(* IEC 61131-3 sources: AXOpen/src/components.ur.robotics/ctrl/src/AxoUrCb3 (part 2) *)

                    Outputs.MotorOn:=_blink.output;

                    IF Inputs.Inputs.Safety.FT_IsFault THEN
                        THIS.CallTimers(FALSE);
                        _power_progress := 310;
                    END_IF;

                    IF Inputs.Inputs.Robot.PW_IsPowerOn THEN
                         Outputs.MotorOn:=FALSE;
                         THIS.CallTimers(FALSE);
                         _power_progress := 321;
                    END_IF;
                END_IF;

                IF _power_progress = 321 THEN
                    TaskMessenger.ActivateOnCondition(ULINT#521, _infoTimer.output, eAxoMessageCategory#Warning);
                    IF _infoTimer.output THEN
                        RobotStatus.Error.Id := UINT#521;
                    END_IF;

                    Outputs.Start:=_blink.output;

                    IF Inputs.Inputs.Safety.FT_IsFault THEN
                        THIS.CallTimers(FALSE);
                        _power_progress := 310;
                    END_IF;

                    IF Inputs.Inputs.Robot.PR_IsProgramRunning AND NOT Inputs.Inputs.Safety.FT_IsFault THEN
                         Outputs.Start:=FALSE;
                         THIS.CallTimers(FALSE);
                         _power_progress := 322;
                    END_IF;
                END_IF;

                IF _power_progress = 322 THEN
                    StartMotorsAndProgramTask.DoneWhen(TRUE);
                    THIS.CallTimers(FALSE);
                    _power_progress := 0;
                END_IF;

                THIS.CallTimers(TRUE);
                StartMotorsAndProgramTask.ThrowWhen(_errorTimer.output);
                RobotStatus.Action.Id := TO_UINT(_power_progress);
            END_IF;
            IF StartMotorsAndProgramTask.DoneReached() THEN
                RobotStatus.Action.Id :=  UINT#111;
                RobotStatus.Error.Id :=  UINT#0;
            ELSIF StartMotorsAndProgramTask.ErrorOccured() THEN
                RobotStatus.Action.Id :=  UINT#810;
                RobotStatus.Error.Id  :=  UINT#810;
            ELSIF StartMotorsAndProgramTask.AbortTriggered() THEN
                RobotStatus.Action.Id :=  UINT#811;
                RobotStatus.Error.Id  :=  UINT#811;
            END_IF;
            Messenger.ActivateOnCondition(ULINT#810,StartMotorsAndProgramTask.HasError(), eAxoMessageCategory#Error);
            Messenger.ActivateOnCondition(ULINT#811,StartMotorsAndProgramTask.IsAborted(), eAxoMessageCategory#Error);
            Messenger.ActivateOnCondition(ULINT#112,StartMotorsAndProgramTask.RestoreTriggered() , eAxoMessageCategory#Error);
            IF StartMotorsAndProgramTask.RestoreTriggered() AND _power_progress >= 310 AND _power_progress <= 329  THEN
                RobotStatus.Action.Id :=  UINT#112;
                _power_progress := 0;
            END_IF;
            //*******************************************

            //***********StartMotorsProgramAndMovementsTask*******
            StartMotorsProgramAndMovementsTask.IsDisabled := _stopTasksAreActive OR StartProgramTask.IsBusy() OR StartMotorsTask.IsBusy() OR StartMovementsTask.IsBusy();
            IF StartMotorsProgramAndMovementsTask.StartTriggered() THEN
                RobotStatus.Action.Id :=  UINT#130;
            END_IF;
            Messenger.ActivateOnCondition(ULINT#130,StartMotorsProgramAndMovementsTask.IsBusy(), eAxoMessageCategory#Info);
            Messenger.ActivateOnCondition(ULINT#131,StartMotorsProgramAndMovementsTask.IsDone(), eAxoMessageCategory#Info);
            IF StartMotorsProgramAndMovementsTask.Execute() THEN
                _blink.Blink(Context := _context, inOnTime:=T#500MS,inOffTime:=T#500MS);

                IF _power_progress = 0 THEN
                    RobotStatus.Error.Id := UINT#0;
                    TaskMessenger.Restore();
                    THIS.CallTimers(FALSE);
                    _power_progress := 330;
                END_IF;

                IF _power_progress = 330 THEN
                    TaskMessenger.ActivateOnCondition(ULINT#530, _infoTimer.output AND NOT Inputs.Inputs.Safety.NO_IsNormalMode, eAxoMessageCategory#Warning);
                    TaskMessenger.ActivateOnCondition(ULINT#531, _infoTimer.output AND NOT Inputs.Inputs.Safety.RD_IsReducedMode, eAxoMessageCategory#Warning);
                    IF _infoTimer.output THEN
                        IF NOT Inputs.Inputs.Safety.NO_IsNormalMode THEN
                            RobotStatus.Error.Id := UINT#530;
                        END_IF;
                        IF NOT Inputs.Inputs.Safety.RD_IsReducedMode THEN
                            RobotStatus.Error.Id := UINT#531;
                        END_IF;
                    END_IF;

                    IF Inputs.Inputs.Safety.NO_IsNormalMode OR Inputs.Inputs.Safety.RD_IsReducedMode THEN
                        THIS.CallTimers(FALSE);
                        _power_progress:=332;
                    END_IF;
                END_IF;

                IF _power_progress = 332 THEN	//Reseting error
                    TaskMessenger.ActivateOnCondition(ULINT#632, _infoTimer.output, eAxoMessageCategory#Warning);
                    IF _infoTimer.output THEN
                        RobotStatus.Error.Id := UINT#632;
                    END_IF;

                    IF NOT Inputs.Inputs.Safety.FT_IsFault THEN
                        THIS.CallTimers(FALSE);
                        _power_progress := 333;
                    END_IF;
                END_IF;

                IF _power_progress = 333 THEN	//Reseting emergency stop error
                    TaskMessenger.ActivateOnCondition(ULINT#533, _infoTimer.output AND Inputs.Inputs.Safety.ES_IsEmergencyStopped , eAxoMessageCategory#Warning);
                    TaskMessenger.ActivateOnCondition(ULINT#534, _infoTimer.output AND Inputs.Inputs.Safety.PS_IsProtectiveStopped , eAxoMessageCategory#Warning);
                    TaskMessenger.ActivateOnCondition(ULINT#535, _infoTimer.output AND Inputs.Inputs.Safety.SS_IsSafeguardStopped , eAxoMessageCategory#Warning);
                    TaskMessenger.ActivateOnCondition(ULINT#536, _infoTimer.output AND Inputs.Inputs.Safety.RC_IsRecoveryMode , eAxoMessageCategory#Warning);
                    TaskMessenger.ActivateOnCondition(ULINT#537, _infoTimer.output AND Inputs.Inputs.Safety.ST_IsStoppedDueSafety , eAxoMessageCategory#Warning);
                    TaskMessenger.ActivateOnCondition(ULINT#538, _infoTimer.output AND Inputs.Inputs.Safety.VL_IsViolation , eAxoMessageCategory#Warning);
                    IF _infoTimer.output THEN
                        IF Inputs.Inputs.Safety.ES_IsEmergencyStopped  THEN
                            RobotStatus.Error.Id := UINT#533;
                        END_IF;
                        IF Inputs.Inputs.Safety.PS_IsProtectiveStopped  THEN
                            RobotStatus.Error.Id := UINT#534;
                        END_IF;
                        IF Inputs.Inputs.Safety.SS_IsSafeguardStopped  THEN
                            RobotStatus.Error.Id := UINT#535;
                        END_IF;
                        IF Inputs.Inputs.Safety.RC_IsRecoveryMode  THEN
                            RobotStatus.Error.Id := UINT#536;
                        END_IF;
                        IF Inputs.Inputs.Safety.ST_IsStoppedDueSafety  THEN
                            RobotStatus.Error.Id := UINT#537;
                        END_IF;
                        IF Inputs.Inputs.Safety.VL_IsViolation  THEN
                            RobotStatus.Error.Id := UINT#538;
                        END_IF;
                    END_IF;

                    IF NOT Inputs.Inputs.Safety.ES_IsEmergencyStopped
                        AND NOT Inputs.Inputs.Safety.PS_IsProtectiveStopped
                        AND NOT Inputs.Inputs.Safety.SS_IsSafeguardStopped
                        AND NOT Inputs.Inputs.Safety.RC_IsRecoveryMode
                        AND NOT Inputs.Inputs.Safety.ST_IsStoppedDueSafety
                        AND NOT Inputs.Inputs.Safety.VL_IsViolation THEN
                        THIS.CallTimers(FALSE);
                        _power_progress := 339;
                    END_IF;
                END_IF;

                IF _power_progress = 339 THEN	//Starting the motors
                    TaskMessenger.ActivateOnCondition(ULINT#539, _infoTimer.output, eAxoMessageCategory#Warning);
                    IF _infoTimer.output THEN
                        RobotStatus.Error.Id := UINT#539;
                    END_IF;

                    Outputs.MotorOn:=_blink.output;

                    IF Inputs.Inputs.Safety.FT_IsFault THEN
                        THIS.CallTimers(FALSE);
                        _power_progress := 330;
                    END_IF;

                    IF Inputs.Inputs.Robot.PW_IsPowerOn AND NOT Inputs.Inputs.Safety.FT_IsFault THEN
                         Outputs.MotorOn:=FALSE;
                         THIS.CallTimers(FALSE);
                         _power_progress := 340;
                    END_IF;
                END_IF;

                IF _power_progress = 340 THEN	// Starting the program
                    TaskMessenger.ActivateOnCondition(ULINT#540, _infoTimer.output, eAxoMessageCategory#Warning);
                    IF _infoTimer.output THEN
                        RobotStatus.Error.Id := UINT#540;
                    END_IF;

                    Outputs.Start:=_blink.output;

                    IF Inputs.Inputs.Safety.FT_IsFault THEN
                        THIS.CallTimers(FALSE);
                        _power_progress := 330;
                    END_IF;

                    IF Inputs.Inputs.Robot.PR_IsProgramRunning AND NOT Inputs.Inputs.Safety.FT_IsFault THEN
                         Outputs.Start:=FALSE;
                         THIS.CallTimers(FALSE);
                         _power_progress := 341;
                    END_IF;
                END_IF;

                IF _power_progress = 341 THEN // Setting the  movement parameters
                    TaskMessenger.ActivateOnCondition(ULINT#541, _infoTimer.output, eAxoMessageCategory#Warning);
                    IF _infoTimer.output THEN
                        RobotStatus.Error.Id := UINT#541;
                    END_IF;
                    Outputs.GlobalSpeed     := TO_DINT(RobotStatus.CurrentMovementParameters.GlobalSpeed);
                    Outputs.ToolNo          := TO_DINT(RobotStatus.CurrentMovementParameters.ToolNo);
                    Outputs.WorkobjectNo    := TO_DINT(RobotStatus.CurrentMovementParameters.WorkobjectNo);
                    Outputs.PointNo         := TO_DINT(RobotStatus.CurrentMovementParameters.PointNo);
                    Outputs.UserSpecSpeed1  := RobotStatus.CurrentMovementParameters.UserSpecSpeed1;
                    Outputs.UserSpecSpeed2  := RobotStatus.CurrentMovementParameters.UserSpecSpeed2;
                    Outputs.Coordinates     := RobotStatus.CurrentMovementParameters.Coordinates;

                    Outputs.ActionNo := DINT#254;

                    IF Outputs.ActionNo = Inputs.ActionNo THEN
                        THIS.CallTimers(FALSE);
                        _power_progress := 342;
                    END_IF;
                END_IF;

                IF _power_progress = 342 THEN //Comparing the movement parameters.
                    TaskMessenger.ActivateOnCondition(ULINT#542, _infoTimer.output AND Inputs.GlobalSpeed <> TO_DINT(RobotStatus.CurrentMovementParameters.GlobalSpeed), eAxoMessageCategory#Warning);
                    TaskMessenger.ActivateOnCondition(ULINT#543, _infoTimer.output AND Inputs.ToolNo <> TO_DINT(RobotStatus.CurrentMovementParameters.ToolNo), eAxoMessageCategory#Warning);
                    TaskMessenger.ActivateOnCondition(ULINT#544, _infoTimer.output AND Inputs.WorkobjectNo <> TO_DINT(RobotStatus.CurrentMovementParameters.WorkobjectNo), eAxoMessageCategory#Warning);
                    TaskMessenger.ActivateOnCondition(ULINT#545, _infoTimer.output AND Inputs.PointNo <> TO_DINT(RobotStatus.CurrentMovementParameters.PointNo), eAxoMessageCategory#Warning);
                    TaskMessenger.ActivateOnCondition(ULINT#546, _infoTimer.output AND Inputs.UserSpecSpeed1 <> RobotStatus.CurrentMovementParameters.UserSpecSpeed1, eAxoMessageCategory#Warning);
                    TaskMessenger.ActivateOnCondition(ULINT#547, _infoTimer.output AND Inputs.UserSpecSpeed2 <> RobotStatus.CurrentMovementParameters.UserSpecSpeed2, eAxoMessageCategory#Warning);
                    IF _infoTimer.output THEN
                        IF Inputs.GlobalSpeed <> TO_DINT(RobotStatus.CurrentMovementParameters.GlobalSpeed) THEN
                            RobotStatus.Error.Id := UINT#542;//<#Waiting for Inputs.GlobalSpeed to be equal to MovementParameters.GlobalSpeed!
                        END_IF;
                        IF Inputs.ToolNo <> TO_DINT(RobotStatus.CurrentMovementParameters.ToolNo) THEN
                            RobotStatus.Error.Id := UINT#543;//<#Waiting for Inputs.ToolNo to be equal to MovementParameters.ToolNo!
                        END_IF;
                        IF Inputs.WorkobjectNo <> TO_DINT(RobotStatus.CurrentMovementParameters.WorkobjectNo) THEN
                            RobotStatus.Error.Id := UINT#544;//<#Waiting for Inputs.WorkobjectNo to be equal to MovementParameters.WorkobjectNo!
                        END_IF;
                        IF Inputs.PointNo <> TO_DINT(RobotStatus.CurrentMovementParameters.PointNo) THEN
                            RobotStatus.Error.Id := UINT#545;//<#Waiting for Inputs.PointNo to be equal to MovementParameters.PointNo!
                        END_IF;
                        IF Inputs.UserSpecSpeed1 <> RobotStatus.CurrentMovementParameters.UserSpecSpeed1 THEN
                            RobotStatus.Error.Id := UINT#546;//<#Waiting for Inputs.UserSpecSpeed1 to be equal to MovementParameters.UserSpecSpeed1!
                        END_IF;
                        IF Inputs.UserSpecSpeed2 <> RobotStatus.CurrentMovementParameters.UserSpecSpeed2 THEN
                            RobotStatus.Error.Id := UINT#547;//<#Waiting for Inputs.UserSpecSpeed2 to be equal to MovementParameters.UserSpecSpeed2!
                        END_IF;
                    END_IF;

                    IF 	Inputs.GlobalSpeed      = TO_DINT(RobotStatus.CurrentMovementParameters.GlobalSpeed) AND
                        Inputs.ToolNo           = TO_DINT(RobotStatus.CurrentMovementParameters.ToolNo) AND
                        Inputs.WorkobjectNo     = TO_DINT(RobotStatus.CurrentMovementParameters.WorkobjectNo) AND
                        Inputs.PointNo          = TO_DINT(RobotStatus.CurrentMovementParameters.PointNo) AND
                        Inputs.UserSpecSpeed1   = RobotStatus.CurrentMovementParameters.UserSpecSpeed1 AND
                        Inputs.UserSpecSpeed2   = RobotStatus.CurrentMovementParameters.UserSpecSpeed2 AND
                        AXOpen.Components.Robotics.CoordinatesAreNearlyEqual(Inputs.Coordinates,RobotStatus.CurrentMovementParameters.Coordinates,REAL#0.01,REAL#0.01,REAL#0.01,REAL#0.01,REAL#0.01,REAL#0.01) THEN
                        THIS.CallTimers(FALSE);
                        _power_progress:=348;
                    END_IF;
                END_IF;

                IF _power_progress = 348 THEN //Acknowledging the movement parameters
                    TaskMessenger.ActivateOnCondition(ULINT#548, _infoTimer.output, eAxoMessageCategory#Warning);
                    IF _infoTimer.output THEN
                        RobotStatus.Error.Id := UINT#548;
                    END_IF;

                    Outputs.ActionNo := DINT#255;

                    IF Outputs.ActionNo = Inputs.ActionNo THEN
                        THIS.CallTimers(FALSE);
                        _power_progress:=349;
                    END_IF;
                END_IF;

                IF _power_progress = 349 THEN
                    TaskMessenger.ActivateOnCondition(ULINT#549, _infoTimer.output, eAxoMessageCategory#Warning);
                    IF _infoTimer.output THEN
                        RobotStatus.Error.Id := UINT#549;
                    END_IF;

                    Outputs.ActionNo := TO_DINT(RobotStatus.CurrentMovementParameters.ActionNo);

                    IF Outputs.ActionNo = Inputs.ActionNo THEN
                        THIS.CallTimers(FALSE);
                        _power_progress:=350;
                    END_IF;
                END_IF;

                IF _power_progress = 350 THEN
                    TaskMessenger.ActivateOnCondition(ULINT#550, _infoTimer.output, eAxoMessageCategory#Warning);
                    IF _infoTimer.output THEN
                        RobotStatus.Error.Id := UINT#550;
                    END_IF;

                    Outputs.ActionNo := DINT#255;

                    IF Outputs.ActionNo = Inputs.ActionNo THEN
                        _power_progress := 0;
                        StartMotorsProgramAndMovementsTask.DoneWhen(TRUE);
                    END_IF;
                END_IF;

	            THIS.CallTimers(TRUE);
                StartMotorsProgramAndMovementsTask.ThrowWhen(_errorTimer.output);
                RobotStatus.Action.Id := TO_UINT(_power_progress);
            END_IF;
            IF StartMotorsProgramAndMovementsTask.DoneReached() THEN
                RobotStatus.Action.Id :=  UINT#131;
                RobotStatus.Error.Id :=  UINT#0;
            ELSIF StartMotorsProgramAndMovementsTask.ErrorOccured() THEN
                RobotStatus.Action.Id :=  UINT#830;
                RobotStatus.Error.Id  :=  UINT#830;
            ELSIF StartMotorsProgramAndMovementsTask.AbortTriggered() THEN
                RobotStatus.Action.Id :=  UINT#831;
                RobotStatus.Error.Id  :=  UINT#831;
            END_IF;
            Messenger.ActivateOnCondition(ULINT#830,StartMotorsProgramAndMovementsTask.HasError(), eAxoMessageCategory#Error);
            Messenger.ActivateOnCondition(ULINT#831,StartMotorsProgramAndMovementsTask.IsAborted(), eAxoMessageCategory#Error);
            Messenger.ActivateOnCondition(ULINT#132,StartMotorsProgramAndMovementsTask.RestoreTriggered() , eAxoMessageCategory#Error);
            IF StartMotorsProgramAndMovementsTask.RestoreTriggered() AND _power_progress >= 330 AND _power_progress <= 359 THEN
                RobotStatus.Action.Id :=  UINT#132;
                _power_progress := 0;
            END_IF;
            //*******************************************

            //***********StartMotorsTask*****************
            StartMotorsTask.IsDisabled := _stopTasksAreActive OR StartMotorsProgramAndMovementsTask.IsBusy() OR StartMotorsAndProgramTask.IsBusy();
            IF StartMotorsTask.StartTriggered() THEN
                RobotStatus.Action.Id :=  UINT#160;
            END_IF;
            Messenger.ActivateOnCondition(ULINT#160,StartMotorsTask.IsBusy(), eAxoMessageCategory#Info);
            Messenger.ActivateOnCondition(ULINT#161,StartMotorsTask.IsDone(), eAxoMessageCategory#Info);
            IF StartMotorsTask.Execute() THEN
                _blink.Blink(Context := _context, inOnTime:=T#500MS,inOffTime:=T#500MS);

                IF _power_progress = 0 THEN
                    RobotStatus.Error.Id := UINT#0;
                    TaskMessenger.Restore();
                    THIS.CallTimers(FALSE);
                    _power_progress := 360;
                END_IF;

                IF _power_progress = 360 THEN
                    TaskMessenger.ActivateOnCondition(ULINT#560, _infoTimer.output AND NOT Inputs.Inputs.Safety.NO_IsNormalMode, eAxoMessageCategory#Warning);
                    TaskMessenger.ActivateOnCondition(ULINT#561, _infoTimer.output AND NOT Inputs.Inputs.Safety.RD_IsReducedMode, eAxoMessageCategory#Warning);
                    IF _infoTimer.output THEN
                        IF NOT Inputs.Inputs.Safety.NO_IsNormalMode THEN
                            RobotStatus.Error.Id := UINT#560;
                        END_IF;
                        IF NOT Inputs.Inputs.Safety.RD_IsReducedMode THEN
                            RobotStatus.Error.Id := UINT#561;
                        END_IF;
                    END_IF;

                    IF Inputs.Inputs.Safety.NO_IsNormalMode OR Inputs.Inputs.Safety.RD_IsReducedMode THEN
                        THIS.CallTimers(FALSE);
                        _power_progress:=362;
                    END_IF;

                END_IF;

                IF _power_progress = 362 THEN	//Reseting error
                    TaskMessenger.ActivateOnCondition(ULINT#562, _infoTimer.output, eAxoMessageCategory#Warning);

                    IF _infoTimer.output THEN
                        RobotStatus.Error.Id := UINT#562;
                    END_IF;

                    IF NOT Inputs.Inputs.Safety.FT_IsFault THEN
                        THIS.CallTimers(FALSE);
                        _power_progress := 363;
                    END_IF;
                END_IF;

                IF _power_progress = 363 THEN	//Reseting emergency stop error

                    TaskMessenger.ActivateOnCondition(ULINT#563, _infoTimer.output AND Inputs.Inputs.Safety.ES_IsEmergencyStopped , eAxoMessageCategory#Warning);
                    TaskMessenger.ActivateOnCondition(ULINT#564, _infoTimer.output AND Inputs.Inputs.Safety.PS_IsProtectiveStopped , eAxoMessageCategory#Warning);
                    TaskMessenger.ActivateOnCondition(ULINT#565, _infoTimer.output AND Inputs.Inputs.Safety.SS_IsSafeguardStopped , eAxoMessageCategory#Warning);
                    TaskMessenger.ActivateOnCondition(ULINT#566, _infoTimer.output AND Inputs.Inputs.Safety.RC_IsRecoveryMode , eAxoMessageCategory#Warning);
                    TaskMessenger.ActivateOnCondition(ULINT#567, _infoTimer.output AND Inputs.Inputs.Safety.ST_IsStoppedDueSafety , eAxoMessageCategory#Warning);
                    TaskMessenger.ActivateOnCondition(ULINT#568, _infoTimer.output AND Inputs.Inputs.Safety.VL_IsViolation , eAxoMessageCategory#Warning);
                    IF _infoTimer.output THEN
                        IF Inputs.Inputs.Safety.ES_IsEmergencyStopped  THEN
                            RobotStatus.Error.Id := UINT#563;
                        END_IF;
                        IF Inputs.Inputs.Safety.PS_IsProtectiveStopped  THEN
                            RobotStatus.Error.Id := UINT#564;
                        END_IF;
                        IF Inputs.Inputs.Safety.SS_IsSafeguardStopped  THEN
                            RobotStatus.Error.Id := UINT#565;
                        END_IF;
                        IF Inputs.Inputs.Safety.RC_IsRecoveryMode  THEN
                            RobotStatus.Error.Id := UINT#566;
                        END_IF;
                        IF Inputs.Inputs.Safety.ST_IsStoppedDueSafety  THEN
                            RobotStatus.Error.Id := UINT#567;
                        END_IF;
                        IF Inputs.Inputs.Safety.VL_IsViolation  THEN
                            RobotStatus.Error.Id := UINT#568;
                        END_IF;
                    END_IF;

                    IF NOT Inputs.Inputs.Safety.ES_IsEmergencyStopped
                        AND NOT Inputs.Inputs.Safety.PS_IsProtectiveStopped
                        AND NOT Inputs.Inputs.Safety.SS_IsSafeguardStopped
                        AND NOT Inputs.Inputs.Safety.RC_IsRecoveryMode
                        AND NOT Inputs.Inputs.Safety.ST_IsStoppedDueSafety
                        AND NOT Inputs.Inputs.Safety.VL_IsViolation THEN
                        THIS.CallTimers(FALSE);
                        _power_progress := 369;
                    END_IF;
                END_IF;

                IF _power_progress = 369 THEN
                    TaskMessenger.ActivateOnCondition(ULINT#569, _infoTimer.output AND NOT Inputs.Inputs.Robot.PW_IsPowerOn, eAxoMessageCategory#Warning);
                    TaskMessenger.ActivateOnCondition(ULINT#570, _infoTimer.output AND Inputs.Inputs.Safety.FT_IsFault, eAxoMessageCategory#Warning);
                    TaskMessenger.ActivateOnCondition(ULINT#571, _infoTimer.output AND Inputs.Inputs.Joints.JointMode_0 <> 253 , eAxoMessageCategory#Warning);
                    TaskMessenger.ActivateOnCondition(ULINT#572, _infoTimer.output AND Inputs.Inputs.Joints.JointMode_1 <> 253 , eAxoMessageCategory#Warning);
                    TaskMessenger.ActivateOnCondition(ULINT#573, _infoTimer.output AND Inputs.Inputs.Joints.JointMode_2 <> 253 , eAxoMessageCategory#Warning);
                    TaskMessenger.ActivateOnCondition(ULINT#574, _infoTimer.output AND Inputs.Inputs.Joints.JointMode_3 <> 253 , eAxoMessageCategory#Warning);
                    TaskMessenger.ActivateOnCondition(ULINT#575, _infoTimer.output AND Inputs.Inputs.Joints.JointMode_4 <> 253 , eAxoMessageCategory#Warning);
                    TaskMessenger.ActivateOnCondition(ULINT#576, _infoTimer.output AND Inputs.Inputs.Joints.JointMode_5 <> 253 , eAxoMessageCategory#Warning);

                    IF _infoTimer.output THEN
                        IF NOT Inputs.Inputs.Robot.PW_IsPowerOn THEN
                            RobotStatus.Error.Id := UINT#569;
                        END_IF;
                        IF Inputs.Inputs.Safety.FT_IsFault  THEN
                            RobotStatus.Error.Id := UINT#570;
                        END_IF;
                        IF Inputs.Inputs.Joints.JointMode_0 <> 253  THEN
                            RobotStatus.Error.Id := UINT#571;
                        END_IF;
                        IF Inputs.Inputs.Joints.JointMode_1 <> 253  THEN
                            RobotStatus.Error.Id := UINT#572;
                        END_IF;
                        IF Inputs.Inputs.Joints.JointMode_2 <> 253  THEN
                            RobotStatus.Error.Id := UINT#573;
                        END_IF;
                        IF Inputs.Inputs.Joints.JointMode_3 <> 253  THEN
                            RobotStatus.Error.Id := UINT#574;
                        END_IF;
                        IF Inputs.Inputs.Joints.JointMode_4 <> 253  THEN
                            RobotStatus.Error.Id := UINT#575;
                        END_IF;
                        IF Inputs.Inputs.Joints.JointMode_5 <> 253  THEN
                            RobotStatus.Error.Id := UINT#576;
                        END_IF;
                    END_IF;

                    Outputs.MotorOn:=_blink.output;

                    IF Inputs.Inputs.Safety.FT_IsFault THEN
                        THIS.CallTimers(FALSE);
                        _power_progress := 360;
                    END_IF;

                    IF Inputs.Inputs.Robot.PW_IsPowerOn AND NOT Inputs.Inputs.Safety.FT_IsFault  AND
                        Inputs.Inputs.Joints.JointMode_0 = 253 AND
                        Inputs.Inputs.Joints.JointMode_1 = 253 AND
                        Inputs.Inputs.Joints.JointMode_2 = 253 AND
                        Inputs.Inputs.Joints.JointMode_3 = 253 AND
                        Inputs.Inputs.Joints.JointMode_4 = 253 AND
                        Inputs.Inputs.Joints.JointMode_5 = 253 THEN
                         Outputs.MotorOn:=FALSE;
                         THIS.CallTimers(FALSE);
                         _power_progress := 377;
                    END_IF;
                END_IF;

                IF _power_progress = 377 THEN
                    StartMotorsTask.DoneWhen(TRUE);
                    THIS.CallTimers(FALSE);
                    _power_progress := 0;
                END_IF;

                THIS.CallTimers(TRUE);
                StartMotorsTask.ThrowWhen(_errorTimer.output);
                RobotStatus.Action.Id := TO_UINT(_power_progress);
            END_IF;
            IF StartMotorsTask.IsFirstExecutionCycle() THEN
                MovementParameters := RobotStatus.CurrentMovementParameters;
            END_IF;
            IF StartMotorsTask.DoneReached() THEN
                RobotStatus.Action.Id :=  UINT#161;
                RobotStatus.Error.Id :=  UINT#0;
            ELSIF StartMotorsTask.ErrorOccured() THEN
                RobotStatus.Action.Id :=  UINT#860;
                RobotStatus.Error.Id  :=  UINT#860;
            ELSIF StartMotorsTask.AbortTriggered() THEN
                RobotStatus.Action.Id :=  UINT#861;
                RobotStatus.Error.Id  :=  UINT#861;
            END_IF;
            Messenger.ActivateOnCondition(ULINT#860,StartMotorsTask.HasError(), eAxoMessageCategory#Error);
            Messenger.ActivateOnCondition(ULINT#861,StartMotorsTask.IsAborted(), eAxoMessageCategory#Error);
            Messenger.ActivateOnCondition(ULINT#162,StartMotorsTask.RestoreTriggered() , eAxoMessageCategory#Error);
            IF StartMotorsTask.RestoreTriggered() AND _power_progress >= 360 AND _power_progress <= 379 THEN
                RobotStatus.Action.Id :=  UINT#162;
                _power_progress := 0;
            END_IF;

            //*******************************************

            //***********StartMovementsTask**************
            StartMovementsTask.IsDisabled := _stopTasksAreActive OR StartMotorsProgramAndMovementsTask.IsBusy();
            IF StartMovementsTask.StartTriggered() THEN
                RobotStatus.Action.Id :=  UINT#180;
            END_IF;
            Messenger.ActivateOnCondition(ULINT#180,StartMovementsTask.IsBusy(), eAxoMessageCategory#Info);
            Messenger.ActivateOnCondition(ULINT#181,StartMovementsTask.IsDone(), eAxoMessageCategory#Info);
            IF StartMovementsTask.Execute() THEN
                IF _movement_progress = 0 THEN
                    RobotStatus.Error.Id :=  UINT#0;
                    TaskMessenger.Restore();
                    THIS.CallTimers(FALSE);
                    _movement_progress := 380;
                END_IF;

                IF _movement_progress = 380 THEN
                    TaskMessenger.ActivateOnCondition(ULINT#580, _infoTimer.output, eAxoMessageCategory#Warning);
                    IF _infoTimer.output THEN
                        RobotStatus.Error.Id := UINT#580;
                    END_IF;

                    IF Inputs.Inputs.Robot.PR_IsProgramRunning THEN
                        THIS.CallTimers(FALSE);
                        _movement_progress := 381;
                    END_IF;
                END_IF;

                IF _movement_progress = 381 THEN
                    TaskMessenger.ActivateOnCondition(ULINT#581, _infoTimer.output, eAxoMessageCategory#Warning);
                    IF _infoTimer.output THEN
                        RobotStatus.Error.Id := UINT#581;
                    END_IF;

                    IF Inputs.Inputs.Robot.PW_IsPowerOn THEN
                        THIS.CallTimers(FALSE);
                        _movement_progress := 382;
                    END_IF;
                END_IF;

                IF _movement_progress = 382 THEN
                    TaskMessenger.ActivateOnCondition(ULINT#582, _infoTimer.output, eAxoMessageCategory#Warning);
                    IF _infoTimer.output THEN
                        RobotStatus.Error.Id := UINT#582;
                    END_IF;

                    IF NOT Inputs.Inputs.Safety.FT_IsFault THEN
                        THIS.CallTimers(FALSE);
                        _movement_progress := 383;
                    END_IF;
                END_IF;

                IF _movement_progress = 383 THEN
                    TaskMessenger.ActivateOnCondition(ULINT#583, _infoTimer.output, eAxoMessageCategory#Warning);
                    IF _infoTimer.output THEN
                        RobotStatus.Error.Id := UINT#583;
                    END_IF;

                    Outputs.GlobalSpeed     := TO_DINT(RobotStatus.CurrentMovementParameters.GlobalSpeed);
                    Outputs.ToolNo          := TO_DINT(RobotStatus.CurrentMovementParameters.ToolNo);
                    Outputs.WorkobjectNo    := TO_DINT(RobotStatus.CurrentMovementParameters.WorkobjectNo);
                    Outputs.PointNo         := TO_DINT(RobotStatus.CurrentMovementParameters.PointNo);
                    Outputs.UserSpecSpeed1  := RobotStatus.CurrentMovementParameters.UserSpecSpeed1;
                    Outputs.UserSpecSpeed2  := RobotStatus.CurrentMovementParameters.UserSpecSpeed2;
                    Outputs.Coordinates     := RobotStatus.CurrentMovementParameters.Coordinates;

                    Outputs.ActionNo := DINT#254;

                    IF Outputs.ActionNo = Inputs.ActionNo THEN
                        THIS.CallTimers(FALSE);
                        _power_progress := 384;
                    END_IF;
                END_IF;

                IF _power_progress = 384 THEN
                    TaskMessenger.ActivateOnCondition(ULINT#584, _infoTimer.output AND Inputs.GlobalSpeed <> TO_DINT(RobotStatus.CurrentMovementParameters.GlobalSpeed), eAxoMessageCategory#Warning);
                    TaskMessenger.ActivateOnCondition(ULINT#585, _infoTimer.output AND Inputs.ToolNo <> TO_DINT(RobotStatus.CurrentMovementParameters.ToolNo), eAxoMessageCategory#Warning);
                    TaskMessenger.ActivateOnCondition(ULINT#586, _infoTimer.output AND Inputs.WorkobjectNo <> TO_DINT(RobotStatus.CurrentMovementParameters.WorkobjectNo) , eAxoMessageCategory#Warning);
                    TaskMessenger.ActivateOnCondition(ULINT#587, _infoTimer.output AND Inputs.PointNo <> TO_DINT(RobotStatus.CurrentMovementParameters.PointNo) , eAxoMessageCategory#Warning);
                    TaskMessenger.ActivateOnCondition(ULINT#588, _infoTimer.output AND Inputs.UserSpecSpeed1 <> RobotStatus.CurrentMovementParameters.UserSpecSpeed1 , eAxoMessageCategory#Warning);
                    TaskMessenger.ActivateOnCondition(ULINT#589, _infoTimer.output AND Inputs.UserSpecSpeed2 <> RobotStatus.CurrentMovementParameters.UserSpecSpeed2, eAxoMessageCategory#Warning);

                    IF _infoTimer.output THEN
                        IF Inputs.GlobalSpeed <> TO_DINT(RobotStatus.CurrentMovementParameters.GlobalSpeed) THEN
                            RobotStatus.Error.Id := UINT#584;//<#Waiting for Inputs.GlobalSpeed to be equal to MovementParameters.GlobalSpeed!
                        END_IF;
                        IF Inputs.ToolNo <> TO_DINT(RobotStatus.CurrentMovementParameters.ToolNo) THEN
                            RobotStatus.Error.Id := UINT#585;//<#Waiting for Inputs.ToolNo to be equal to MovementParameters.ToolNo!
                        END_IF;
                        IF Inputs.WorkobjectNo <> TO_DINT(RobotStatus.CurrentMovementParameters.WorkobjectNo) THEN
                            RobotStatus.Error.Id := UINT#586;//<#Waiting for Inputs.WorkobjectNo to be equal to MovementParameters.WorkobjectNo!
                        END_IF;
                        IF Inputs.PointNo <> TO_DINT(RobotStatus.CurrentMovementParameters.PointNo) THEN
                            RobotStatus.Error.Id := UINT#587;//<#Waiting for Inputs.PointNo to be equal to MovementParameters.PointNo!
                        END_IF;
                        IF Inputs.UserSpecSpeed1 <> RobotStatus.CurrentMovementParameters.UserSpecSpeed1 THEN
                            RobotStatus.Error.Id := UINT#588;//<#Waiting for Inputs.UserSpecSpeed1 to be equal to MovementParameters.UserSpecSpeed1!
                        END_IF;
                        IF Inputs.UserSpecSpeed2 <> RobotStatus.CurrentMovementParameters.UserSpecSpeed2 THEN
                            RobotStatus.Error.Id := UINT#589;//<#Waiting for Inputs.UserSpecSpeed2 to be equal to MovementParameters.UserSpecSpeed2!
                        END_IF;
                    END_IF;

                    IF 	Inputs.GlobalSpeed      = TO_DINT(RobotStatus.CurrentMovementParameters.GlobalSpeed) AND
                        Inputs.ToolNo           = TO_DINT(RobotStatus.CurrentMovementParameters.ToolNo) AND
                        Inputs.WorkobjectNo     = TO_DINT(RobotStatus.CurrentMovementParameters.WorkobjectNo) AND
                        Inputs.PointNo          = TO_DINT(RobotStatus.CurrentMovementParameters.PointNo) AND
                        Inputs.UserSpecSpeed1   = RobotStatus.CurrentMovementParameters.UserSpecSpeed1 AND
                        Inputs.UserSpecSpeed2   = RobotStatus.CurrentMovementParameters.UserSpecSpeed2 AND
                        AXOpen.Components.Robotics.CoordinatesAreNearlyEqual(Inputs.Coordinates,RobotStatus.CurrentMovementParameters.Coordinates,REAL#0.01,REAL#0.01,REAL#0.01,REAL#0.01,REAL#0.01,REAL#0.01) THEN
                        THIS.CallTimers(FALSE);
                        _movement_progress:=390;
                    END_IF;
                END_IF;

                IF _movement_progress = 390 THEN
                    TaskMessenger.ActivateOnCondition(ULINT#590, _infoTimer.output, eAxoMessageCategory#Warning);
                    IF _infoTimer.output THEN
                        RobotStatus.Error.Id := UINT#590;
                    END_IF;

                    Outputs.ActionNo := DINT#255;

                    IF Outputs.ActionNo = Inputs.ActionNo THEN
                        THIS.CallTimers(FALSE);
                        _movement_progress:=391;
                    END_IF;
                END_IF;

                IF _movement_progress = 391 THEN
                    TaskMessenger.ActivateOnCondition(ULINT#591, _infoTimer.output, eAxoMessageCategory#Warning);
                    IF _infoTimer.output THEN
                        RobotStatus.Error.Id := UINT#591;
                    END_IF;

                    Outputs.ActionNo := TO_DINT(RobotStatus.CurrentMovementParameters.ActionNo);

                    IF Outputs.ActionNo = Inputs.ActionNo THEN
                        THIS.CallTimers(FALSE);
                        _movement_progress:=392;
                    END_IF;
                END_IF;

                IF _movement_progress = 392 THEN
                    TaskMessenger.ActivateOnCondition(ULINT#692, _infoTimer.output, eAxoMessageCategory#Warning);
                    IF _infoTimer.output THEN
                        RobotStatus.Error.Id := UINT#692;
                    END_IF;

                    Outputs.ActionNo := DINT#255;

                    IF Outputs.ActionNo = Inputs.ActionNo THEN
                        _movement_progress := 0;
                        StartMovementsTask.DoneWhen(TRUE);
                    END_IF;
                END_IF;

	            THIS.CallTimers(TRUE);

                StartMovementsTask.ThrowWhen(_errorTimer.output);

                RobotStatus.Action.Id := TO_UINT(_movement_progress);
            END_IF;
            IF StartMovementsTask.DoneReached() THEN
                RobotStatus.Action.Id :=  UINT#181;
                RobotStatus.Error.Id :=  UINT#0;
            ELSIF StartMovementsTask.ErrorOccured() THEN
                RobotStatus.Action.Id :=  UINT#880;
                RobotStatus.Error.Id  :=  UINT#880;
            ELSIF StartMovementsTask.AbortTriggered()THEN
                RobotStatus.Action.Id :=  UINT#881;
                RobotStatus.Error.Id  :=  UINT#881;
            END_IF;
            Messenger.ActivateOnCondition(ULINT#880,StartMovementsTask.HasError(), eAxoMessageCategory#Error);
            Messenger.ActivateOnCondition(ULINT#881,StartMovementsTask.IsAborted(), eAxoMessageCategory#Error);
            Messenger.ActivateOnCondition(ULINT#182,StartMovementsTask.RestoreTriggered() , eAxoMessageCategory#Error);
            IF StartMovementsTask.RestoreTriggered() AND _movement_progress >= 380 AND _movement_progress <= 399  THEN
                RobotStatus.Action.Id :=  UINT#182;
                _movement_progress := 0;
            END_IF;

            //*******************************************

            //***********StartProgramTask*******
            StartProgramTask.IsDisabled := _stopTasksAreActive;
            IF StartProgramTask.StartTriggered() THEN
                RobotStatus.Action.Id :=  UINT#200;
            END_IF;
            Messenger.ActivateOnCondition(ULINT#200,StartProgramTask.IsBusy(), eAxoMessageCategory#Info);
            Messenger.ActivateOnCondition(ULINT#201,StartProgramTask.IsDone(), eAxoMessageCategory#Info);
             IF StartProgramTask.Execute() THEN
                _blink.Blink(Context := _context, inOnTime:=T#500MS,inOffTime:=T#500MS);

                IF _power_progress = 0 THEN
                    RobotStatus.Error.Id :=  UINT#0;
                    TaskMessenger.Restore();
                    THIS.CallTimers(FALSE);
                    _power_progress := 400;
                END_IF;

                IF _power_progress = 400 THEN
                    TaskMessenger.ActivateOnCondition(ULINT#600, _infoTimer.output AND NOT Inputs.Inputs.Safety.NO_IsNormalMode, eAxoMessageCategory#Warning);
                    TaskMessenger.ActivateOnCondition(ULINT#601, _infoTimer.output AND NOT Inputs.Inputs.Safety.RD_IsReducedMode, eAxoMessageCategory#Warning);
                    IF _infoTimer.output THEN
                        IF NOT Inputs.Inputs.Safety.NO_IsNormalMode THEN
                            RobotStatus.Error.Id := UINT#600;
                        END_IF;
                        IF NOT Inputs.Inputs.Safety.RD_IsReducedMode THEN
                            RobotStatus.Error.Id := UINT#601;
                        END_IF;
                    END_IF;

                    IF Inputs.Inputs.Safety.NO_IsNormalMode OR Inputs.Inputs.Safety.RD_IsReducedMode THEN
                        THIS.CallTimers(FALSE);
                        _power_progress:=402;
                    END_IF;
                END_IF;

                IF _power_progress = 402 THEN
                    TaskMessenger.ActivateOnCondition(ULINT#602, _infoTimer.output, eAxoMessageCategory#Warning);
                    IF _infoTimer.output THEN
                        RobotStatus.Error.Id := UINT#602;
                    END_IF;

                    Outputs.Start:=_blink.output;

                    IF Inputs.Inputs.Robot.PR_IsProgramRunning THEN
                         Outputs.Start:=FALSE;
                         THIS.CallTimers(FALSE);
                         _power_progress := 403;
                    END_IF;
                END_IF;

                IF _power_progress = 403 THEN
                    StartProgramTask.DoneWhen(TRUE);
                    THIS.CallTimers(FALSE);
                    _power_progress := 0;
                END_IF;

                THIS.CallTimers(TRUE);
                StartProgramTask.ThrowWhen(_errorTimer.output);
                RobotStatus.Action.Id := TO_UINT(_power_progress);
            END_IF;
            IF StartProgramTask.DoneReached() THEN
                RobotStatus.Action.Id :=  UINT#201;
                RobotStatus.Error.Id :=  UINT#0;
            ELSIF StartProgramTask.ErrorOccured() THEN
                RobotStatus.Action.Id :=  UINT#900;
                RobotStatus.Error.Id  :=  UINT#900;
            ELSIF StartProgramTask.AbortTriggered()THEN
                RobotStatus.Action.Id :=  UINT#901;
                RobotStatus.Error.Id  :=  UINT#901;
            END_IF;
            Messenger.ActivateOnCondition(ULINT#900,StartProgramTask.HasError(), eAxoMessageCategory#Error);
            Messenger.ActivateOnCondition(ULINT#901,StartProgramTask.IsAborted(), eAxoMessageCategory#Error);
            Messenger.ActivateOnCondition(ULINT#202,StartProgramTask.RestoreTriggered() , eAxoMessageCategory#Error);
            IF StartProgramTask.RestoreTriggered() AND _power_progress >= 400 AND _power_progress <= 409  THEN
                RobotStatus.Action.Id :=  UINT#202;
                _power_progress := 0;
            END_IF;
            //*******************************************

            //***********StopMovementsAndProgramTask*****
            StopMovementsAndProgramTask.IsDisabled := FALSE;
            IF StopMovementsAndProgramTask.StartTriggered() THEN
                RobotStatus.Action.Id :=  UINT#210;
            END_IF;
            Messenger.ActivateOnCondition(ULINT#210,StopMovementsAndProgramTask.IsBusy(), eAxoMessageCategory#Info);
            Messenger.ActivateOnCondition(ULINT#211,StopMovementsAndProgramTask.IsDone(), eAxoMessageCategory#Info);
            IF StopMovementsAndProgramTask.Execute() THEN
                IF _power_progress = 0 THEN
                    RobotStatus.Error.Id :=  UINT#0;
                    TaskMessenger.Restore();
                    THIS.CallTimers(FALSE);
                    _power_progress := 410;
                END_IF;

                IF _power_progress = 410 THEN
                    TaskMessenger.ActivateOnCondition(ULINT#610, _infoTimer.output AND NOT Inputs.Inputs.Safety.NO_IsNormalMode, eAxoMessageCategory#Warning);
                    TaskMessenger.ActivateOnCondition(ULINT#611, _infoTimer.output AND NOT Inputs.Inputs.Safety.RD_IsReducedMode, eAxoMessageCategory#Warning);
                    IF _infoTimer.output THEN
                        IF NOT Inputs.Inputs.Safety.NO_IsNormalMode THEN
                            RobotStatus.Error.Id := UINT#610;
                        END_IF;
                        IF NOT Inputs.Inputs.Safety.RD_IsReducedMode THEN
                            RobotStatus.Error.Id := UINT#611;
                        END_IF;
                    END_IF;

                    IF Inputs.Inputs.Safety.NO_IsNormalMode OR Inputs.Inputs.Safety.RD_IsReducedMode THEN
                        THIS.CallTimers(FALSE);
                        _power_progress:=412;
                    END_IF;
                END_IF;

                IF _power_progress = 412 THEN
                    TaskMessenger.ActivateOnCondition(ULINT#612, _infoTimer.output, eAxoMessageCategory#Warning);
                    IF _infoTimer.output THEN
                        RobotStatus.Error.Id := UINT#612;
                    END_IF;

                    Outputs.Stop := TRUE;

                    IF NOT Inputs.Inputs.Robot.PR_IsProgramRunning THEN
                        Outputs.Stop := FALSE ;
                        THIS.CallTimers(FALSE);
                        _power_progress:=413;
                    END_IF;
                END_IF;

                IF _power_progress = 413 THEN
                    Outputs.Pause := FALSE ;
                    StopMovementsAndProgramTask.DoneWhen(TRUE);
                    _power_progress := 0;
                END_IF;

                THIS.CallTimers(TRUE);

                StopMovementsAndProgramTask.ThrowWhen(_errorTimer.output);

                RobotStatus.Action.Id := TO_UINT(_power_progress);
            END_IF;
            IF StopMovementsAndProgramTask.DoneReached() THEN
                RobotStatus.Action.Id :=  UINT#211;
                RobotStatus.Error.Id :=  UINT#0;
            ELSIF StopMovementsAndProgramTask.ErrorOccured() THEN
                RobotStatus.Action.Id :=  UINT#910;
                RobotStatus.Error.Id  :=  UINT#910;
            ELSIF StopMovementsAndProgramTask.AbortTriggered()THEN
                RobotStatus.Action.Id :=  UINT#911;
                RobotStatus.Error.Id  :=  UINT#911;
            END_IF;
            Messenger.ActivateOnCondition(ULINT#910,StopMovementsAndProgramTask.HasError(), eAxoMessageCategory#Error);
            Messenger.ActivateOnCondition(ULINT#911,StopMovementsAndProgramTask.IsAborted(), eAxoMessageCategory#Error);
            Messenger.ActivateOnCondition(ULINT#212,StopMovementsAndProgramTask.RestoreTriggered() , eAxoMessageCategory#Error);
            IF StopMovementsAndProgramTask.RestoreTriggered() AND _power_progress >= 410 AND _power_progress <= 419  THEN
                RobotStatus.Action.Id :=  UINT#212;
                _power_progress := 0;
            END_IF;
            //*******************************************

            //***********StopMovementsTask***************
            StopMovementsTask.IsDisabled := FALSE;
            IF StopMovementsAndProgramTask.StartTriggered() THEN
                RobotStatus.Action.Id :=  UINT#220;
            END_IF;
            Messenger.ActivateOnCondition(ULINT#220,StopMovementsAndProgramTask.IsBusy(), eAxoMessageCategory#Info);
            Messenger.ActivateOnCondition(ULINT#221,StopMovementsAndProgramTask.IsDone(), eAxoMessageCategory#Info);
            IF StopMovementsTask.Execute() THEN
                IF _power_progress = 0 THEN
                    RobotStatus.Error.Id :=  UINT#0;
                    TaskMessenger.Restore();
                    THIS.CallTimers(FALSE);
                    _power_progress := 420;
                END_IF;

                IF _power_progress = 420 THEN
                    TaskMessenger.ActivateOnCondition(ULINT#620, _infoTimer.output AND NOT Inputs.Inputs.Safety.NO_IsNormalMode, eAxoMessageCategory#Warning);
                    TaskMessenger.ActivateOnCondition(ULINT#621, _infoTimer.output AND NOT Inputs.Inputs.Safety.RD_IsReducedMode, eAxoMessageCategory#Warning);
                    IF _infoTimer.output THEN
                        IF NOT Inputs.Inputs.Safety.NO_IsNormalMode THEN
                            RobotStatus.Error.Id := UINT#620;
                        END_IF;
                        IF NOT Inputs.Inputs.Safety.RD_IsReducedMode THEN
                            RobotStatus.Error.Id := UINT#621;
                        END_IF;
                    END_IF;

                    IF Inputs.Inputs.Safety.NO_IsNormalMode OR Inputs.Inputs.Safety.RD_IsReducedMode THEN
                        THIS.CallTimers(FALSE);
                        _power_progress:=422;
                    END_IF;
                END_IF;
                IF _power_progress = 422 THEN
                    TaskMessenger.ActivateOnCondition(ULINT#622, _infoTimer.output, eAxoMessageCategory#Warning);
                    IF _infoTimer.output THEN
                        RobotStatus.Error.Id := UINT#622;
                    END_IF;

                    Outputs.Pause := TRUE;

                    IF NOT Inputs.Inputs.Robot.PR_IsProgramRunning THEN
                        Outputs.Pause := FALSE ;
                        THIS.CallTimers(FALSE);
                        _power_progress:=423;
                    END_IF;
                END_IF;

                IF _power_progress = 423 THEN
                    Outputs.Pause := FALSE ;
                    StopMovementsTask.DoneWhen(TRUE);
                    _power_progress := 0;
                END_IF;
                THIS.CallTimers(TRUE);

                StopMovementsTask.ThrowWhen(_errorTimer.output);

                RobotStatus.Action.Id := TO_UINT(_power_progress);
            END_IF;
            IF StopMovementsTask.DoneReached() THEN
                RobotStatus.Action.Id :=  UINT#221;
                RobotStatus.Error.Id :=  UINT#0;
            ELSIF StopMovementsTask.ErrorOccured() THEN
                RobotStatus.Action.Id :=  UINT#920;
                RobotStatus.Error.Id  :=  UINT#920;
            ELSIF StopMovementsTask.AbortTriggered()THEN
                RobotStatus.Action.Id :=  UINT#921;
                RobotStatus.Error.Id  :=  UINT#921;
            END_IF;
            Messenger.ActivateOnCondition(ULINT#920,StopMovementsTask.HasError(), eAxoMessageCategory#Error);
            Messenger.ActivateOnCondition(ULINT#921,StopMovementsTask.IsAborted(), eAxoMessageCategory#Error);
            Messenger.ActivateOnCondition(ULINT#222,StopMovementsTask.RestoreTriggered() , eAxoMessageCategory#Error);
            IF StopMovementsTask.RestoreTriggered() AND _power_progress >= 420 AND _power_progress <= 429  THEN
                RobotStatus.Action.Id :=  UINT#222;
                _power_progress := 0;
            END_IF;
            //*******************************************

            //***********StopProgramTask*****************
            StopProgramTask.IsDisabled := FALSE;
            IF StopProgramTask.StartTriggered() THEN
                RobotStatus.Action.Id :=  UINT#230;
            END_IF;
            Messenger.ActivateOnCondition(ULINT#230,StopProgramTask.IsBusy(), eAxoMessageCategory#Info);
            Messenger.ActivateOnCondition(ULINT#231,StopProgramTask.IsDone(), eAxoMessageCategory#Info);
            IF StopProgramTask.Execute() THEN
                IF _power_progress = 0 THEN
                    RobotStatus.Error.Id :=  UINT#0;
                    TaskMessenger.Restore();
                    THIS.CallTimers(FALSE);
                    _power_progress := 430;
                END_IF;

                IF _power_progress = 430 THEN
                    TaskMessenger.ActivateOnCondition(ULINT#630, _infoTimer.output AND NOT Inputs.Inputs.Safety.NO_IsNormalMode, eAxoMessageCategory#Warning);
                    TaskMessenger.ActivateOnCondition(ULINT#631, _infoTimer.output AND NOT Inputs.Inputs.Safety.RD_IsReducedMode, eAxoMessageCategory#Warning);

                    IF _infoTimer.output THEN
                        IF NOT Inputs.Inputs.Safety.NO_IsNormalMode THEN
                            RobotStatus.Error.Id := UINT#630;
                        END_IF;
                        IF NOT Inputs.Inputs.Safety.RD_IsReducedMode THEN
                            RobotStatus.Error.Id := UINT#631;
                        END_IF;
                    END_IF;

                    IF Inputs.Inputs.Safety.NO_IsNormalMode OR Inputs.Inputs.Safety.RD_IsReducedMode THEN
                        THIS.CallTimers(FALSE);
                        _power_progress:=432;
                    END_IF;
                END_IF;

                IF _power_progress = 432 THEN
                    TaskMessenger.ActivateOnCondition(ULINT#632, _infoTimer.output, eAxoMessageCategory#Warning);
                    IF _infoTimer.output THEN
                        RobotStatus.Error.Id := UINT#632;
                    END_IF;

                    Outputs.Stop := TRUE;

                    IF NOT Inputs.Inputs.Robot.PR_IsProgramRunning THEN
                        Outputs.Stop := FALSE ;
                        THIS.CallTimers(FALSE);
                        _power_progress:=433;
                    END_IF;
                END_IF;

                IF _power_progress = 433 THEN
                    Outputs.Pause := FALSE ;
                    StopProgramTask.DoneWhen(TRUE);
                    _power_progress := 0;
                END_IF;

                THIS.CallTimers(TRUE);

                StopProgramTask.ThrowWhen(_errorTimer.output);

                RobotStatus.Action.Id := TO_UINT(_power_progress);
            END_IF;
            IF StopProgramTask.DoneReached() THEN
                RobotStatus.Action.Id :=  UINT#231;
                RobotStatus.Error.Id :=  UINT#0;
            ELSIF StopProgramTask.ErrorOccured() THEN
                RobotStatus.Action.Id :=  UINT#930;
                RobotStatus.Error.Id  :=  UINT#930;
            ELSIF StopProgramTask.AbortTriggered()THEN
                RobotStatus.Action.Id :=  UINT#931;
                RobotStatus.Error.Id  :=  UINT#931;
            END_IF;
            Messenger.ActivateOnCondition(ULINT#930,StopProgramTask.HasError(), eAxoMessageCategory#Error);
            Messenger.ActivateOnCondition(ULINT#931,StopProgramTask.IsAborted(), eAxoMessageCategory#Error);
            Messenger.ActivateOnCondition(ULINT#232,StopProgramTask.RestoreTriggered() , eAxoMessageCategory#Error);
            IF StopProgramTask.RestoreTriggered() AND _power_progress >= 430 AND _power_progress <= 439  THEN
                RobotStatus.Action.Id :=  UINT#232;
                _power_progress := 0;
            END_IF;

            //*******************************************

            //*************POWER ON********************
            PowerOnTask.IsDisabled := NOT(Inputs.RobotMode=eAxoUrRoboticsRobotMode#DISCONNECTED AND Config.RemotePowerOnEnabled);
            IF PowerOnTask.Execute() THEN
                refPowerOnPulse^ :=TRUE;
                RobotStatus.Action.Id :=  UINT#420;//('<#POWER ON PULSE WAS SEND TO CONTROLER#>');
                PowerOnTask.DoneWhen(PowerOnTask.Duration > Config.RemotePowerOnPulse);
            END_IF;

            IF refPowerOnPulse^ AND PowerOnTask.IsDone()  OR NOT Config.RemotePowerOnEnabled THEN
                refPowerOnPulse^ :=FALSE;
            END_IF;

            //****************************************

            _someTaskIsActive := StartAtMainTask.IsBusy()
                                OR StartMotorsAndProgramTask.IsBusy()
                                OR StartMovementsTask.IsBusy()
                                OR StartMovementsTask.IsBusy()
                                OR StopMovementsTask.IsBusy()
                                OR StopMovementsAndProgramTask.IsBusy()
                                OR StopProgramTask.IsBusy();

            Messenger.ActivateOnCondition(ULINT#719,_someTaskIsActive AND Inputs.Inputs.Safety.ES_IsEmergencyStopped, eAxoMessageCategory#Error);
            Messenger.ActivateOnCondition(ULINT#720,_someTaskIsActive AND Inputs.Inputs.Safety.ST_IsStoppedDueSafety, eAxoMessageCategory#Error);

            IF _someTaskIsActive THEN
                IF(Inputs.Inputs.Safety.ES_IsEmergencyStopped) THEN
                    RobotStatus.Error.Id := UINT#719;
                END_IF;
                IF(Inputs.Inputs.Safety.ST_IsStoppedDueSafety) THEN
                    RobotStatus.Error.Id := UINT#720;
                END_IF;
            END_IF;
            //***********UPDATE**OUTPUTS*****************
            //SYSTEM OUTPUTS
            Outputs.Outputs.Reg1.Bit_0 := Outputs.Start;
            Outputs.outputs.Reg1.Bit_1 := Outputs.Stop;
            Outputs.outputs.Reg1.Bit_2 := Outputs.Pause;
            Outputs.outputs.Reg1.Bit_3 := Outputs.MotorOn;
            //Outputs.outputs.Reg1.Bit_4 := Outputs.RunAction;

            //Tool signals
            Outputs.Outputs.Reg1.Bit_8 := Outputs.Tool_1_Retract;
            Outputs.outputs.Reg1.Bit_9 := Outputs.Tool_1_Extend;
            Outputs.outputs.Reg1.Bit_10 := Outputs.Tool_2_Retract;
            Outputs.outputs.Reg1.Bit_11 := Outputs.Tool_2_Extend;
            Outputs.outputs.Reg1.Bit_12 := Outputs.Tool_3_Retract;
            Outputs.outputs.Reg1.Bit_13 := Outputs.Tool_3_Extend;
            Outputs.outputs.Reg1.Bit_14 := Outputs.Tool_4_Retract;
            Outputs.outputs.Reg1.Bit_15 := Outputs.Tool_4_Extend;

            //zone
            Outputs.Outputs.Reg1.Int_0 := Outputs.Zone;
            //position
            Outputs.Outputs.Reg1.Int_1 := Outputs.InPosition;

            //Movement parameters
            Outputs.Outputs.Reg1.Int_2 := Outputs.ActionNo;
            Outputs.Outputs.Reg1.Int_3 := Outputs.GlobalSpeed;
            Outputs.Outputs.Reg1.Int_4 := Outputs.ToolNo;
            Outputs.Outputs.Reg1.Int_5 := Outputs.WorkobjectNo;
            Outputs.Outputs.Reg1.Int_6 := Outputs.PointNo;
            //master mode  such as manual/auto ....
            Outputs.Outputs.Reg1.Int_7 := TO_DINT(Outputs.MasterMode);

            Outputs.Outputs.Reg1.Float_0 := Outputs.UserSpecSpeed1;
            Outputs.Outputs.Reg1.Float_1 := Outputs.UserSpecSpeed2;

            ////Coordinates
            Outputs.Outputs.Reg1.Float_2 := Outputs.Coordinates.X ;
            Outputs.Outputs.Reg1.Float_3 := Outputs.Coordinates.Y;
            Outputs.Outputs.Reg1.Float_4 := Outputs.Coordinates.Z ;
            Outputs.Outputs.Reg1.Float_5 := (Outputs.Coordinates.Rx);
            Outputs.Outputs.Reg1.Float_6 := (Outputs.Coordinates.Ry);
            Outputs.Outputs.Reg1.Float_7 := (Outputs.Coordinates.Rz);

            //st_URO_CB3_O2TSpeedData => 8_O2T Robot IO
            _data24[0].%X0 := Outputs.Outputs.Speed.SSM_SpeedSliderFractionMask;

            _dword := TO_DWORD(Outputs.Outputs.Speed.SpeedSliderFraction * REAL#0.01);
            _data24[4] := _dword.%B3;
            _data24[5] := _dword.%B2;
            _data24[6] := _dword.%B1;
            _data24[7] := _dword.%B0;

            //st_URO_CB3_O2TIoData => 8_O2T Robot IO
            _data24[8]  := TO_BYTE(Outputs.Outputs.IO.StandardDigitalOutputMask);
            _data24[9]  := TO_BYTE(Outputs.Outputs.IO.ConfigurableDigitalOutputMask);
            _data24[10] := TO_BYTE(Outputs.Outputs.IO.StandardDigitalOutputs);
            _data24[11] := TO_BYTE(Outputs.Outputs.IO.ConfigurableDdigitalOutputs);
            _data24[12] := TO_BYTE(Outputs.Outputs.IO.AOM_AnalogOutputMask);
            _data24[13] := TO_BYTE(Outputs.Outputs.IO.AOT_AnalogOutputTypes);
            _data24[14] := TO_BYTE(Outputs.Outputs.IO.TDOM_ToolDigitalOutputMask);
            _data24[15] := TO_BYTE(Outputs.Outputs.IO.TDO_ToolDigitalOutput);

            _dword := TO_DWORD(Outputs.Outputs.IO.StandardAnalogOutput_0);
            _data24[16] := _dword.%B3;
            _data24[17] := _dword.%B2;
            _data24[18] := _dword.%B1;
            _data24[19] := _dword.%B0;

            _dword := TO_DWORD(Outputs.Outputs.IO.StandardAnalogOutput_1);
            _data24[20] := _dword.%B3;
            _data24[21] := _dword.%B2;
            _data24[22] := _dword.%B1;
            _data24[23] := _dword.%B0;

            returnValue := Siemens.Simatic.S71500.DistributedIO.WriteData(_hwIdAxoUrRobotics_O2T_Robot_IO,_data24);
            Messenger.ActivateOnCondition(ULINT#721,returnValue > WORD#0, eAxoMessageCategory#ProgrammingError);
            IF returnValue > WORD#0 THEN
                RobotStatus.Error.Id := UINT#721;
                RETURN;
            END_IF;

            //st_URO_CB3_O2TRegData => 9_O2T General Purpose Registers 1
            _data100[0].%X0 :=  Outputs.Outputs.Reg1.Bit_0;
            _data100[0].%X1 :=  Outputs.Outputs.Reg1.Bit_1;
            _data100[0].%X2 :=  Outputs.Outputs.Reg1.Bit_2;
            _data100[0].%X3 :=  Outputs.Outputs.Reg1.Bit_3;
            _data100[0].%X4 :=  Outputs.Outputs.Reg1.Bit_4;
            _data100[0].%X5 :=  Outputs.Outputs.Reg1.Bit_5;
            _data100[0].%X6 :=  Outputs.Outputs.Reg1.Bit_6;
            _data100[0].%X7 :=  Outputs.Outputs.Reg1.Bit_7;

            _data100[1].%X0 :=  Outputs.Outputs.Reg1.Bit_8;
            _data100[1].%X1 :=  Outputs.Outputs.Reg1.Bit_9;
            _data100[1].%X2 :=  Outputs.Outputs.Reg1.Bit_10;
            _data100[1].%X3 :=  Outputs.Outputs.Reg1.Bit_11;
            _data100[1].%X4 :=  Outputs.Outputs.Reg1.Bit_12;
            _data100[1].%X5 :=  Outputs.Outputs.Reg1.Bit_13;
            _data100[1].%X6 :=  Outputs.Outputs.Reg1.Bit_14;
            _data100[1].%X7 :=  Outputs.Outputs.Reg1.Bit_15;

            _data100[2].%X0 :=  Outputs.Outputs.Reg1.Bit_16;
            _data100[2].%X1 :=  Outputs.Outputs.Reg1.Bit_17;
            _data100[2].%X2 :=  Outputs.Outputs.Reg1.Bit_18;
            _data100[2].%X3 :=  Outputs.Outputs.Reg1.Bit_19;
            _data100[2].%X4 :=  Outputs.Outputs.Reg1.Bit_20;
            _data100[2].%X5 :=  Outputs.Outputs.Reg1.Bit_21;
            _data100[2].%X6 :=  Outputs.Outputs.Reg1.Bit_22;
            _data100[2].%X7 :=  Outputs.Outputs.Reg1.Bit_23;

            _data100[3].%X0 :=  Outputs.Outputs.Reg1.Bit_24;
            _data100[3].%X1 :=  Outputs.Outputs.Reg1.Bit_25;
            _data100[3].%X2 :=  Outputs.Outputs.Reg1.Bit_26;
            _data100[3].%X3 :=  Outputs.Outputs.Reg1.Bit_27;
            _data100[3].%X4 :=  Outputs.Outputs.Reg1.Bit_28;
            _data100[3].%X5 :=  Outputs.Outputs.Reg1.Bit_29;
            _data100[3].%X6 :=  Outputs.Outputs.Reg1.Bit_30;
            _data100[3].%X7 :=  Outputs.Outputs.Reg1.Bit_31;

            _dword          := TO_DWORD( Outputs.Outputs.Reg1.Int_0);
            _data100[4]     := _dword.%B3;
            _data100[5]     := _dword.%B2;
            _data100[6]     := _dword.%B1;
            _data100[7]     := _dword.%B0;

            _dword          := TO_DWORD( Outputs.Outputs.Reg1.Int_1);
            _data100[8]     := _dword.%B3;
            _data100[9]     := _dword.%B2;
            _data100[10]    := _dword.%B1;
            _data100[11]    := _dword.%B0;

            _dword          := TO_DWORD( Outputs.Outputs.Reg1.Int_2);
            _data100[12]    := _dword.%B3;
            _data100[13]    := _dword.%B2;
            _data100[14]    := _dword.%B1;
            _data100[15]    := _dword.%B0;

            _dword          := TO_DWORD( Outputs.Outputs.Reg1.Int_3);
            _data100[16]    := _dword.%B3;
            _data100[17]    := _dword.%B2;
            _data100[18]    := _dword.%B1;
            _data100[19]    := _dword.%B0;

            _dword          := TO_DWORD( Outputs.Outputs.Reg1.Int_4);
            _data100[20]    := _dword.%B3;
            _data100[21]    := _dword.%B2;
            _data100[22]    := _dword.%B1;
            _data100[23]    := _dword.%B0;

            _dword          := TO_DWORD( Outputs.Outputs.Reg1.Int_5);
            _data100[24]    := _dword.%B3;
            _data100[25]    := _dword.%B2;
            _data100[26]    := _dword.%B1;
            _data100[27]    := _dword.%B0;

            _dword          := TO_DWORD( Outputs.Outputs.Reg1.Int_6);
            _data100[28]    := _dword.%B3;
            _data100[29]    := _dword.%B2;
            _data100[30]    := _dword.%B1;
            _data100[31]    := _dword.%B0;

            _dword          := TO_DWORD( Outputs.Outputs.Reg1.Int_7);
            _data100[32]    := _dword.%B3;
            _data100[33]    := _dword.%B2;
            _data100[34]    := _dword.%B1;
            _data100[35]    := _dword.%B0;

            _dword          := TO_DWORD( Outputs.Outputs.Reg1.Int_8);
            _data100[36]    := _dword.%B3;
            _data100[37]    := _dword.%B2;
            _data100[38]    := _dword.%B1;
            _data100[39]    := _dword.%B0;

            _dword          := TO_DWORD( Outputs.Outputs.Reg1.Int_9);
            _data100[40]    := _dword.%B3;
            _data100[41]    := _dword.%B2;
            _data100[42]    := _dword.%B1;
            _data100[43]    := _dword.%B0;

            _dword          := TO_DWORD( Outputs.Outputs.Reg1.Int_10);
            _data100[44]    := _dword.%B3;
            _data100[45]    := _dword.%B2;
            _data100[46]    := _dword.%B1;
            _data100[47]    := _dword.%B0;

            _dword          := TO_DWORD( Outputs.Outputs.Reg1.Int_11);
            _data100[48]    := _dword.%B3;
            _data100[49]    := _dword.%B2;
            _data100[50]    := _dword.%B1;
            _data100[51]    := _dword.%B0;

            _dword          := TO_DWORD( Outputs.Outputs.Reg1.Float_0);
            _data100[52]    := _dword.%B3;
            _data100[53]    := _dword.%B2;
            _data100[54]    := _dword.%B1;
            _data100[55]    := _dword.%B0;

            _dword          := TO_DWORD( Outputs.Outputs.Reg1.Float_1);
            _data100[56]    := _dword.%B3;
            _data100[58]    := _dword.%B2;
            _data100[58]    := _dword.%B1;
            _data100[59]    := _dword.%B0;

            _dword          := TO_DWORD( Outputs.Outputs.Reg1.Float_2);
            _data100[60]    := _dword.%B3;
            _data100[61]    := _dword.%B2;
            _data100[62]    := _dword.%B1;
            _data100[63]    := _dword.%B0;

            _dword          := TO_DWORD( Outputs.Outputs.Reg1.Float_3);
            _data100[64]    := _dword.%B3;
            _data100[65]    := _dword.%B2;
            _data100[66]    := _dword.%B1;
            _data100[67]    := _dword.%B0;

            _dword          := TO_DWORD( Outputs.Outputs.Reg1.Float_4);
            _data100[68]    := _dword.%B3;
            _data100[69]    := _dword.%B2;
            _data100[70]    := _dword.%B1;
            _data100[71]    := _dword.%B0;

            _dword          := TO_DWORD( Outputs.Outputs.Reg1.Float_5);
            _data100[72]    := _dword.%B3;
            _data100[73]    := _dword.%B2;
            _data100[74]    := _dword.%B1;
            _data100[75]    := _dword.%B0;

            _dword          := TO_DWORD( Outputs.Outputs.Reg1.Float_6);
            _data100[76]    := _dword.%B3;
            _data100[77]    := _dword.%B2;
            _data100[78]    := _dword.%B1;
            _data100[79]    := _dword.%B0;

            _dword          := TO_DWORD( Outputs.Outputs.Reg1.Float_7);
            _data100[80]    := _dword.%B3;
            _data100[81]    := _dword.%B2;
            _data100[82]    := _dword.%B1;
            _data100[83]    := _dword.%B0;

            _dword          := TO_DWORD( Outputs.Outputs.Reg1.Float_8);
            _data100[84]    := _dword.%B3;
            _data100[85]    := _dword.%B2;
            _data100[86]    := _dword.%B1;
            _data100[87]    := _dword.%B0;

            _dword          := TO_DWORD( Outputs.Outputs.Reg1.Float_9);
            _data100[88]    := _dword.%B3;
            _data100[89]    := _dword.%B2;
            _data100[90]    := _dword.%B1;
            _data100[91]    := _dword.%B0;

            _dword          := TO_DWORD( Outputs.Outputs.Reg1.Float_10);
            _data100[92]    := _dword.%B3;
            _data100[93]    := _dword.%B2;
            _data100[94]    := _dword.%B1;
            _data100[95]    := _dword.%B0;

            _dword          := TO_DWORD( Outputs.Outputs.Reg1.Float_11);
            _data100[96]    := _dword.%B3;
            _data100[97]    := _dword.%B2;
            _data100[98]    := _dword.%B1;
            _data100[99]    := _dword.%B0;

            returnValue := Siemens.Simatic.S71500.DistributedIO.WriteData(_hwIdAxoUrRobotics_O2T_General_Purpose_Registers_1,_data100);
            Messenger.ActivateOnCondition(ULINT#722,returnValue > WORD#0, eAxoMessageCategory#ProgrammingError);
            IF returnValue > WORD#0 THEN
                RobotStatus.Error.Id := UINT#722;
                RETURN;
            END_IF;

            //st_URO_CB3_O2TRegData => 10_O2T General Purpose Registers 2
            _data100[0].%X0 :=  Outputs.Outputs.Reg2.Bit_0;
            _data100[0].%X1 :=  Outputs.Outputs.Reg2.Bit_1;
            _data100[0].%X2 :=  Outputs.Outputs.Reg2.Bit_2;
            _data100[0].%X3 :=  Outputs.Outputs.Reg2.Bit_3;
            _data100[0].%X4 :=  Outputs.Outputs.Reg2.Bit_4;
            _data100[0].%X5 :=  Outputs.Outputs.Reg2.Bit_5;
            _data100[0].%X6 :=  Outputs.Outputs.Reg2.Bit_6;
            _data100[0].%X7 :=  Outputs.Outputs.Reg2.Bit_7;

            _data100[1].%X0 :=  Outputs.Outputs.Reg2.Bit_8;
            _data100[1].%X1 :=  Outputs.Outputs.Reg2.Bit_9;
            _data100[1].%X2 :=  Outputs.Outputs.Reg2.Bit_10;
            _data100[1].%X3 :=  Outputs.Outputs.Reg2.Bit_11;
            _data100[1].%X4 :=  Outputs.Outputs.Reg2.Bit_12;
            _data100[1].%X5 :=  Outputs.Outputs.Reg2.Bit_13;
            _data100[1].%X6 :=  Outputs.Outputs.Reg2.Bit_14;
            _data100[1].%X7 :=  Outputs.Outputs.Reg2.Bit_15;

            _data100[2].%X0 :=  Outputs.Outputs.Reg2.Bit_16;
            _data100[2].%X1 :=  Outputs.Outputs.Reg2.Bit_17;
            _data100[2].%X2 :=  Outputs.Outputs.Reg2.Bit_18;
            _data100[2].%X3 :=  Outputs.Outputs.Reg2.Bit_19;
            _data100[2].%X4 :=  Outputs.Outputs.Reg2.Bit_20;
            _data100[2].%X5 :=  Outputs.Outputs.Reg2.Bit_21;
            _data100[2].%X6 :=  Outputs.Outputs.Reg2.Bit_22;
            _data100[2].%X7 :=  Outputs.Outputs.Reg2.Bit_23;

            _data100[3].%X0 :=  Outputs.Outputs.Reg2.Bit_24;
            _data100[3].%X1 :=  Outputs.Outputs.Reg2.Bit_25;
            _data100[3].%X2 :=  Outputs.Outputs.Reg2.Bit_26;
            _data100[3].%X3 :=  Outputs.Outputs.Reg2.Bit_27;
            _data100[3].%X4 :=  Outputs.Outputs.Reg2.Bit_28;
            _data100[3].%X5 :=  Outputs.Outputs.Reg2.Bit_29;
            _data100[3].%X6 :=  Outputs.Outputs.Reg2.Bit_30;
            _data100[3].%X7 :=  Outputs.Outputs.Reg2.Bit_31;

            _dword          := TO_DWORD( Outputs.Outputs.Reg2.Int_0);
            _data100[4]     := _dword.%B3;
            _data100[5]     := _dword.%B2;
            _data100[6]     := _dword.%B1;
            _data100[7]     := _dword.%B0;

            _dword          := TO_DWORD( Outputs.Outputs.Reg2.Int_1);
            _data100[8]     := _dword.%B3;
            _data100[9]     := _dword.%B2;
            _data100[10]    := _dword.%B1;
            _data100[11]    := _dword.%B0;

            _dword          := TO_DWORD( Outputs.Outputs.Reg2.Int_2);
            _data100[12]    := _dword.%B3;
            _data100[13]    := _dword.%B2;
            _data100[14]    := _dword.%B1;
            _data100[15]    := _dword.%B0;

            _dword          := TO_DWORD( Outputs.Outputs.Reg2.Int_3);
            _data100[16]    := _dword.%B3;
            _data100[17]    := _dword.%B2;
            _data100[18]    := _dword.%B1;
            _data100[19]    := _dword.%B0;

            _dword          := TO_DWORD( Outputs.Outputs.Reg2.Int_4);
            _data100[20]    := _dword.%B3;
            _data100[21]    := _dword.%B2;
            _data100[22]    := _dword.%B1;
            _data100[23]    := _dword.%B0;

            _dword          := TO_DWORD( Outputs.Outputs.Reg2.Int_5);
            _data100[24]    := _dword.%B3;
            _data100[25]    := _dword.%B2;
            _data100[26]    := _dword.%B1;
            _data100[27]    := _dword.%B0;

            _dword          := TO_DWORD( Outputs.Outputs.Reg2.Int_6);
            _data100[28]    := _dword.%B3;
            _data100[29]    := _dword.%B2;
            _data100[30]    := _dword.%B1;
            _data100[31]    := _dword.%B0;

            _dword          := TO_DWORD( Outputs.Outputs.Reg2.Int_7);
            _data100[32]    := _dword.%B3;
            _data100[33]    := _dword.%B2;
            _data100[34]    := _dword.%B1;
            _data100[35]    := _dword.%B0;

            _dword          := TO_DWORD( Outputs.Outputs.Reg2.Int_8);
            _data100[36]    := _dword.%B3;
            _data100[37]    := _dword.%B2;
            _data100[38]    := _dword.%B1;
            _data100[39]    := _dword.%B0;

            _dword          := TO_DWORD( Outputs.Outputs.Reg2.Int_9);
            _data100[40]    := _dword.%B3;
            _data100[41]    := _dword.%B2;
            _data100[42]    := _dword.%B1;
            _data100[43]    := _dword.%B0;

            _dword          := TO_DWORD( Outputs.Outputs.Reg2.Int_10);
            _data100[44]    := _dword.%B3;
            _data100[45]    := _dword.%B2;
            _data100[46]    := _dword.%B1;
            _data100[47]    := _dword.%B0;

            _dword          := TO_DWORD( Outputs.Outputs.Reg2.Int_11);
            _data100[48]    := _dword.%B3;
            _data100[49]    := _dword.%B2;
            _data100[50]    := _dword.%B1;
            _data100[51]    := _dword.%B0;

            _dword          := TO_DWORD( Outputs.Outputs.Reg2.Float_0);
            _data100[52]    := _dword.%B3;
            _data100[53]    := _dword.%B2;
            _data100[54]    := _dword.%B1;
            _data100[55]    := _dword.%B0;

            _dword          := TO_DWORD( Outputs.Outputs.Reg2.Float_1);
            _data100[56]    := _dword.%B3;
            _data100[58]    := _dword.%B2;
            _data100[58]    := _dword.%B1;
            _data100[59]    := _dword.%B0;

            _dword          := TO_DWORD( Outputs.Outputs.Reg2.Float_2);
            _data100[60]    := _dword.%B3;
            _data100[61]    := _dword.%B2;
            _data100[62]    := _dword.%B1;
            _data100[63]    := _dword.%B0;

            _dword          := TO_DWORD( Outputs.Outputs.Reg2.Float_3);
            _data100[64]    := _dword.%B3;
            _data100[65]    := _dword.%B2;
            _data100[66]    := _dword.%B1;
            _data100[67]    := _dword.%B0;

            _dword          := TO_DWORD( Outputs.Outputs.Reg2.Float_4);
            _data100[68]    := _dword.%B3;
            _data100[69]    := _dword.%B2;
            _data100[70]    := _dword.%B1;
            _data100[71]    := _dword.%B0;

            _dword          := TO_DWORD( Outputs.Outputs.Reg2.Float_5);
            _data100[72]    := _dword.%B3;
            _data100[73]    := _dword.%B2;
            _data100[74]    := _dword.%B1;
            _data100[75]    := _dword.%B0;

            _dword          := TO_DWORD( Outputs.Outputs.Reg2.Float_6);
            _data100[76]    := _dword.%B3;
            _data100[77]    := _dword.%B2;
            _data100[78]    := _dword.%B1;
            _data100[79]    := _dword.%B0;

            _dword          := TO_DWORD( Outputs.Outputs.Reg2.Float_7);
            _data100[80]    := _dword.%B3;
            _data100[81]    := _dword.%B2;
            _data100[82]    := _dword.%B1;
            _data100[83]    := _dword.%B0;

            _dword          := TO_DWORD( Outputs.Outputs.Reg2.Float_8);
            _data100[84]    := _dword.%B3;
            _data100[85]    := _dword.%B2;
            _data100[86]    := _dword.%B1;
            _data100[87]    := _dword.%B0;

            _dword          := TO_DWORD( Outputs.Outputs.Reg2.Float_9);
            _data100[88]    := _dword.%B3;
            _data100[89]    := _dword.%B2;
            _data100[90]    := _dword.%B1;
            _data100[91]    := _dword.%B0;

            _dword          := TO_DWORD( Outputs.Outputs.Reg2.Float_10);
            _data100[92]    := _dword.%B3;
            _data100[93]    := _dword.%B2;
            _data100[94]    := _dword.%B1;
            _data100[95]    := _dword.%B0;

            _dword          := TO_DWORD( Outputs.Outputs.Reg2.Float_11);
            _data100[96]    := _dword.%B3;
            _data100[97]    := _dword.%B2;
            _data100[98]    := _dword.%B1;
            _data100[99]    := _dword.%B0;

            returnValue := Siemens.Simatic.S71500.DistributedIO.WriteData(_hwIdAxoUrRobotics_O2T_General_Purpose_Registers_2,_data100);
            Messenger.ActivateOnCondition(ULINT#723,returnValue > WORD#0, eAxoMessageCategory#ProgrammingError);
            IF returnValue > WORD#0 THEN
                RobotStatus.Error.Id := UINT#723;
                RETURN;
            END_IF;

            //*******************************************
            THIS.Close();
        END_METHOD

        METHOD PROTECTED OVERRIDE ManualControl
            RobotStatus.CurrentMovementParameters := MovementParameters;
        END_METHOD

        ///<summary>
        /// Restores this component into intial state.
        ///</summary>
        METHOD PUBLIC OVERRIDE Restore
            PowerOnTask.Restore();
            StopMovementsTask.Restore();
            StopMovementsAndProgramTask.Restore();
            StopProgramTask.Restore();
            // StopMotorsTask.Restore();
            StartAtMainTask.Restore();
            StartMotorsAndProgramTask.Restore();
            StartProgramTask.Restore();
            StartMotorsTask.Restore();
            StartMovementsTask.Restore();
            StartMotorsProgramAndMovementsTask.Restore();
            RestoreTask.DoneWhen(TRUE);
            _power_progress := 0;
        END_METHOD

        METHOD PUBLIC StartAtMain : IAxoTaskState
            StartAtMain := StartAtMainTask.Invoke();
        END_METHOD

        METHOD PUBLIC StartMotors : IAxoTaskState
            StartMotors := StartMotorsTask.Invoke();
        END_METHOD

        METHOD PUBLIC StartMotorsAndProgram : IAxoTaskState
            StartMotorsAndProgram := StartMotorsAndProgramTask.Invoke();
        END_METHOD

        METHOD PUBLIC StartMotorsProgramAndMovements : IAxoTaskState
            VAR_IN_OUT
                inData : AxoRoboticsMovementsParams;
            END_VAR
            RobotStatus.CurrentMovementParameters := inData;

            StartMotorsProgramAndMovements := StartMotorsProgramAndMovementsTask.Invoke();
        END_METHOD

        METHOD PUBLIC StartMovements : IAxoTaskState
            VAR_IN_OUT
                inData : AxoRoboticsMovementsParams;
            END_VAR
            RobotStatus.CurrentMovementParameters := inData;

            StartMovements := StartMovementsTask.Invoke();
        END_METHOD

        METHOD PUBLIC StartProgram : IAxoTaskState
            StartProgram := StartProgramTask.Invoke();
        END_METHOD

        METHOD PUBLIC StopMovements : IAxoTaskState
            VAR_INPUT
                inStopType : eAxoRoboticsStopType;
            END_VAR
            _stopType := inStopType;
            StopMovements := StopMovementsTask.Invoke();
        END_METHOD

        METHOD PUBLIC StopMovementsAndProgram : IAxoTaskState
            VAR_INPUT
                inStopType : eAxoRoboticsStopType;
            END_VAR
            _stopType := inStopType;
            StopMovementsAndProgram := StopMovementsAndProgramTask.Invoke();
        END_METHOD

        METHOD PUBLIC StopProgram : IAxoTaskState
            StopProgram := StopProgramTask.Invoke();
        END_METHOD

        // METHOD PUBLIC StopMotors : IAxoTaskState
        //     StopMotors := StopMotorsTask.Invoke();
        // END_METHOD

        METHOD PRIVATE CallTimers
            VAR_INPUT
                signal : BOOL;
            END_VAR

            _infoTimer.OnDelay(THIS, signal AND _infoTime > LT#0s , _infoTime);
            _errorTimer.OnDelay(THIS, signal AND _errorTime > LT#0s , _errorTime );
        END_METHOD

        METHOD PRIVATE GetRobotModeDescription : eAxoUrRoboticsRobotMode
            VAR_INPUT
                inMode:USINT;
            END_VAR
            CASE inMode OF
                USINT#0: GetRobotModeDescription := eAxoUrRoboticsRobotMode#DISCONNECTED;
                USINT#1: GetRobotModeDescription := eAxoUrRoboticsRobotMode#SAFETY;
                USINT#2: GetRobotModeDescription := eAxoUrRoboticsRobotMode#BOOTING;
                USINT#3: GetRobotModeDescription := eAxoUrRoboticsRobotMode#POWER_OFF;
                USINT#4: GetRobotModeDescription := eAxoUrRoboticsRobotMode#POWER_ON;
                USINT#5: GetRobotModeDescription := eAxoUrRoboticsRobotMode#IDLE;
                USINT#6: GetRobotModeDescription := eAxoUrRoboticsRobotMode#BACKDRIVE;
                USINT#7: GetRobotModeDescription := eAxoUrRoboticsRobotMode#RUNNING;
                USINT#8: GetRobotModeDescription := eAxoUrRoboticsRobotMode#UPDATING_FIRMWARE;
            END_CASE;
        END_METHOD
    END_CLASS
END_NAMESPACE
